FUNCTION_BLOCK FlushingManager_HMI (* Service Interface Function Block Type *)
  (* Standard: 61499-2 *)
  (* Version 0.0, 6/21/2026, Schneider Electric, template *)
  PACKAGE SE.Nereda;
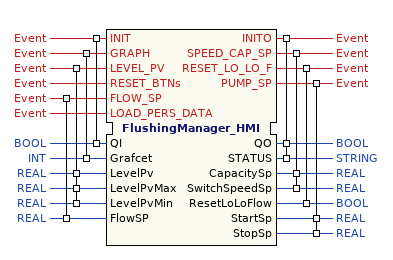
  EVENT_INPUT
    INIT WITH QI;
    GRAPH WITH Grafcet;
    LEVEL_PV WITH LevelPvMax, LevelPvMin, LevelPv;
    RESET_BTNs;
    FLOW_SP WITH FlowSP;
    LOAD_PERS_DATA;
  END_EVENT
  EVENT_OUTPUT
    INITO WITH QO, STATUS;
    SPEED_CAP_SP WITH CapacitySp, SwitchSpeedSp;
    RESET_LO_LO_F WITH ResetLoLoFlow;
    PUMP_SP WITH StartSp, StopSp;
  END_EVENT
  VAR_INPUT
    QI : BOOL;
    Grafcet : INT;
    LevelPv : REAL;
    LevelPvMax : REAL;
    LevelPvMin : REAL;
    FlowSP : REAL;
  END_VAR
  VAR_OUTPUT
    QO : BOOL; (* Event Output Qualifier *)
    STATUS : STRING; (* Service Status *)
    CapacitySp : REAL;
    SwitchSpeedSp : REAL;
    ResetLoLoFlow : BOOL;
    StartSp : REAL;
    StopSp : REAL;
  END_VAR
  SERVICE /
    SEQUENCE 
    END_SEQUENCE
  END_SERVICE
END_FUNCTION_BLOCK
